FUNCTION_BLOCK SkillConfig (* Simple FB with one algorithm *)
  (* Standard: 61499-1 *)
  (* Version 1.0, 2024-07-29, AK123700 *)
  PACKAGE DDBImpl;
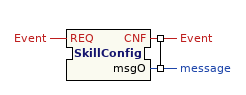
  EVENT_INPUT
    REQ; (* Normal Execution Request *)
  END_EVENT
  EVENT_OUTPUT
    CNF WITH msgO; (* Execution Confirmation *)
  END_EVENT
  VAR_OUTPUT
    msgO : message;
  END_VAR
  EC_STATES
    REQ : REQ -> CNF;
  END_STATES
  ALGORITHM REQ IN ST:

  END_ALGORITHM
END_FUNCTION_BLOCK
